// TIA Portal project "Hotdog Project" (V16)

(* hardware
DEVICE "S7-1200 station_1"  S7-1200 Station
   slot 0: "Rack_0"  S7-1200 Rack  Rack  V1.0
   slot 1: "PLC_1"  CPU 1214C DC/DC/DC  6ES7 214-1AE30-0XB0  V2.0
   slot 3: "AQ 1x12BIT_1"  AQ1 signal board  6ES7 232-4HA30-0XB0  V1.0
*)

// ===== PLC "PLC_1"  CPU 1214C DC/DC/DC =====

VAR_GLOBAL   // PLC tag table "Default tag table"
   "Catsup" AT %I0.0 : Bool;
   "Both" AT %M0.0 : Bool;
   "catsup_rem" AT %M0.1 : Bool;
   "mustard" AT %I0.1 : Bool;
   "mustard_rem" AT %M0.2 : Bool;
END_VAR

// folder: System blocks/Program resources

DATA_BLOCK "Hotdogs"   // DB1
{ S7_Optimized_Access := 'TRUE' }
AUTHOR : Simatic
FAMILY : IEC
NAME : CNTR
VERSION : 1.0
// stored: InstanceOfName IEC_COUNTER
"IEC_COUNTER"
BEGIN
END_DATA_BLOCK

// folder: (top level)

ORGANIZATION_BLOCK "Main"   // OB1, LAD, ProgramCycle
TITLE = "Main Program Sweep (Cycle)"
{ S7_Optimized_Access := 'TRUE' }
VERSION : 0.1
BEGIN

REGION Network 1
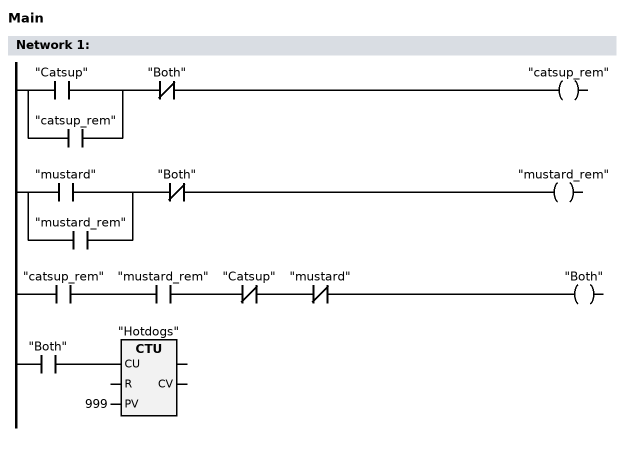
   "catsup_rem" := ("Catsup" OR "catsup_rem") AND NOT "Both";
   "mustard_rem" := ("mustard" OR "mustard_rem") AND NOT "Both";
   "Both" := "catsup_rem" AND "mustard_rem" AND NOT "Catsup" AND NOT "mustard";
   "Hotdogs".CTU(CU := "Both", PV := 999);
END_REGION
END_ORGANIZATION_BLOCK